(* CODESYS project test.export

Project tree, tasks and I/O mapping:
  Device : CODESYS Control Win V3 x64, 3S - Smart Software Solutions GmbH, version 3.5.16.10
    application Application
      libraries: Standard, * (System)
      task MainTask (cyclic, interval 500 ms, priority 1) calls PLC_PRG
      program CFC_TEST [CFC]
      program PLC_PRG [ST]
      program ST_TEST [ST]
*)

// Device/Application/PLC_PRG
PROGRAM PLC_PRG
VAR
END_VAR

CFC_TEST();
ST_TEST();

END_PROGRAM

// Device/Application/CFC_TEST
PROGRAM CFC_TEST
VAR
	A: REAL;
END_VAR

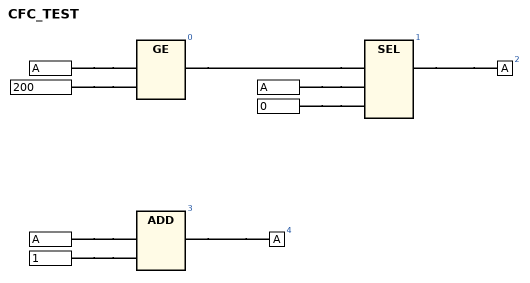
A := SEL(A >= 200, A, 0);
A := A + 1;

END_PROGRAM

// Device/Application/ST_TEST
PROGRAM ST_TEST
VAR
	B: REAL;
END_VAR

IF B>200 THEN
	B:=0;
ELSE
	B:=B+1;
END_IF

END_PROGRAM
